Yaskawa INFORM job: R1_W27-A4(90,180)KM-OK.JBI

/JOB
//NAME R1_W27-A4(90,180)KM-OK
///FOLDERNAME KRIS-SCIANA
//POS
///NPOS 201,201,0,9,0,0
///TOOL 0
///POSTYPE PULSE
///PULSE
C00000=-12408,-168229,-129239,11856,76417,1490
C00001=-114075,-55562,-33330,57879,69757,51049
C00002=-170127,-11218,4712,80761,69619,75034
C00003=-166026,1115,14662,80935,66751,75417
C00004=-166026,1115,14662,80935,66751,75417
C00005=-164179,6139,17196,85884,73779,76491
C00006=-163843,5639,16762,85908,73539,76507
C00007=-164179,6139,17196,85884,73779,76491
C00008=-166496,-467,13337,75702,58764,75189
C00009=-166831,-1552,12436,75705,58996,75152
C00010=-166508,-36,14521,75997,58636,74926
C00011=-166831,-1552,12436,75705,58996,75152
C00012=-166496,-467,13337,75702,58764,75189
C00013=-166021,-3570,934,78534,68009,78358
C00014=-137610,-28929,-19421,69080,47942,64710
C00015=-100776,-35686,-23013,57930,21837,49720
C00016=-103071,-36442,-26491,56591,24205,50318
C00017=-97018,-28630,-27379,22144,28331,59500
C00018=-96530,-21499,-20901,21722,27897,59706
C00019=-100662,-29228,-19206,55793,22319,50751
C00020=-102053,-30601,-20713,56706,23278,50281
C00021=-94207,-25966,-26207,14018,29505,61725
C00022=-90744,-41515,-31094,11154,24096,63148
C00023=-90595,-42140,-31027,11070,23720,63189
C00024=-94073,-53021,-44279,15136,26788,61156
C00025=-105496,-45084,-28829,64380,24182,46446
C00026=-120732,-139011,-128731,13191,-67324,-37746
C00027=-120732,-139011,-128731,13191,-67324,-37746
C00028=-21816,-138429,-128213,9073,25992,-35710
C00029=12937,47891,-35883,-5198,71905,46207
C00030=24559,114456,10111,-12521,95879,79421
C00031=-20060,163701,97232,-14944,96585,79331
C00032=-75754,163701,97232,-14944,96585,79331
C00033=-99437,40505,18804,-2837,35585,35366
C00034=-120732,-117814,-48395,13191,72289,-37746
C00035=-172569,-80041,-34226,-15627,55653,-16743
C00036=-173881,-75690,-28267,-15647,54036,-17014
C00037=-174396,-73921,-25835,-15662,53377,-17117
C00038=-174409,-72642,-23726,-15788,52756,-17025
C00039=-174396,-73921,-25835,-15662,53377,-17117
C00040=-177237,-69247,-20992,-27235,53512,-13633
C00041=-177890,-67562,-19632,-27129,53343,-13864
C00042=-177237,-69247,-20992,-27235,53512,-13633
C00043=-181977,-77418,-24251,-27266,50136,-14704
C00044=-193956,-50227,-14941,539,58562,-29056
C00045=-192915,-50819,-15265,329,58451,-28665
C00046=-194756,-48721,-14111,700,58831,-29355
C00047=-182531,-71466,-31778,-1788,58094,-24759
C00048=-122199,17749,55230,-64618,69888,3761
C00049=-124469,25360,65490,-65961,67496,4502
C00050=-125352,28797,70143,-66592,66515,4877
C00051=-125200,39134,82378,-67427,65683,5911
C00052=-125978,39297,82548,-67654,65232,5820
C00053=-125200,39134,82378,-67427,65683,5911
C00054=-125352,28797,70143,-66592,66515,4877
C00055=-127676,20892,69191,-78285,59026,9362
C00056=-127562,25294,74286,-78756,58894,9826
C00057=-127676,21375,69995,-78428,58968,9490
C00058=-125009,20842,69444,-77518,60577,9664
C00059=-122672,36678,78518,-58027,73309,3381
C00060=-122677,38905,82216,-58303,72687,3837
C00061=-122672,36678,78518,-58027,73309,3381
C00062=-172569,-80041,-34226,-15627,55653,-16743
C00063=-193629,-34313,-13531,-412,84628,-47335
C00064=-193629,-29158,-1725,-414,80010,-47323
C00065=-192771,-30731,-2257,-348,79534,-47037
C00066=-192029,-32324,-3298,-290,79358,-46790
C00067=-192512,-31641,-3367,-327,79748,-46950
C00068=-192512,-32314,-4820,-327,80296,-46951
C00069=-191917,-33584,-5641,-280,80152,-46753
C00070=-191917,-33170,-4750,-280,79815,-46753
C00071=-191917,-35734,-10378,-279,81963,-46757
C00072=-120477,17632,43941,-55533,81040,-704
C00073=-135463,1706,26098,-36401,96659,-64397
C00074=-139240,-2239,32183,-37186,90451,-63806
C00075=-139413,-3608,31065,-37238,90369,-63846
C00076=-139240,-2239,32183,-37186,90451,-63806
C00077=-139240,-982,34590,-37167,89779,-63576
C00078=-139240,-2239,32183,-37186,90451,-63806
C00079=-136968,12512,36999,-36743,95104,-64482
C00080=-139711,-16957,6278,-33197,82477,-62153
C00081=-147688,-28677,-1688,-34006,78458,-64099
C00082=-148352,-29126,-1989,-34060,78161,-64273
C00083=-147688,-28677,-1688,-34006,78458,-64099
C00084=-147688,-29352,-3169,-33950,78930,-64245
C00085=-147969,-31758,-4758,-33997,78605,-64257
C00086=-147969,-31405,-3991,-34026,78361,-64182
C00087=-147969,-31758,-4758,-33997,78605,-64257
C00088=-146343,-30027,-3614,-33855,79395,-63850
C00089=-146343,-29533,-2533,-33893,79050,-63746
C00090=-147651,-30771,-3351,-34009,78431,-64078
C00091=-147340,-30313,-4491,-33895,79336,-64232
C00092=-168861,-24308,-1126,-34250,71707,-70597
C00093=-172727,-20891,3494,-34314,69279,-71427
C00094=-173288,-21050,3382,-34292,69050,-71587
C00095=-172727,-20891,3494,-34314,69279,-71427
C00096=-172727,-21623,1837,-34186,69816,-71602
C00097=-173683,-23699,371,-34172,69302,-71836
C00098=-173683,-23301,1270,-34243,69012,-71740
C00099=-173683,-23699,371,-34172,69302,-71836
C00100=-171105,-22755,1033,-34271,70379,-71106
C00101=-171105,-22220,2243,-34361,69988,-70979
C00102=-172969,-22746,1870,-34294,69220,-71509
C00103=-172838,-23509,-311,-34112,70064,-71727
C00104=-172642,-46434,-14047,-37866,50218,-77712
C00105=-173875,-14141,7002,-35805,52648,-79377
C00106=-177522,-4435,19967,-36117,48708,-79612
C00107=-177904,-4485,19925,-35996,48552,-79746
C00108=-177522,-4435,19967,-36117,48708,-79612
C00109=-177522,-5400,17843,-35709,49372,-79894
C00110=-178274,-6796,17094,-35594,48861,-80070
C00111=-178274,-6447,17863,-35742,48620,-79968
C00112=-178274,-6796,17094,-35594,48861,-80070
C00113=-176755,-6519,17315,-36071,49483,-79541
C00114=-176755,-6106,18226,-36244,49200,-79420
C00115=-177745,-6110,18254,-35943,48780,-79759
C00116=-177557,-6572,16647,-35628,49473,-79954
C00117=-127483,-80419,-25529,-45538,63215,-61268
C00118=-137560,-77057,-18811,-45546,71982,-69050
C00119=-137790,-77163,-18085,-45710,71521,-68929
C00120=-138002,-77837,-18318,-45803,71281,-68907
C00121=-137790,-77163,-18085,-45710,71521,-68929
C00122=-137790,-78839,-20640,-45553,72028,-69171
C00123=-138552,-80734,-20734,-45929,71034,-69027
C00124=-138465,-80152,-20160,-45922,71036,-68989
C00125=-138465,-79547,-19253,-45982,70860,-68902
C00126=-138465,-80152,-20160,-45922,71036,-68989
C00127=-130873,-75354,-22667,-43475,77336,-68607
C00128=-143731,-120291,-35892,-61673,37258,-53156
C00129=-153031,-106896,-24772,-72774,26670,-48341
C00130=-154852,-106645,-24753,-72766,25749,-48792
C00131=-174213,-103200,-24560,-67377,16120,-55832
C00132=-173958,-111624,-32831,-65076,16578,-56845
C00133=-173211,-92844,-38044,-39863,60080,-26099
C00134=-183742,-42639,-8543,-30727,93066,-40842
C00135=-194212,-69823,-30460,-23787,74043,-41412
C00136=-189340,-95494,-32602,-40064,42381,-27057
C00137=-199606,-67555,-26283,-19174,46492,-39002
C00138=-192832,-51591,-10291,-33919,35141,-36541
C00139=-193001,-17027,18379,-39421,24969,-38608
C00140=-185793,-2062,15010,-31452,55489,-48604
C00141=-180914,-39023,-11312,-35464,76884,-35483
C00142=-186493,-28244,-7036,-31408,60621,-50185
C00143=-186186,-25103,-332,-32207,58430,-49503
C00144=-187143,4604,23985,-31838,53193,-48465
C00145=-185793,-2062,15010,-31452,55489,-48604
C00146=-188015,-40449,-12502,-32039,52292,-48508
C00147=-190017,-70687,-28062,-34017,46482,-47362
C00148=-197564,-65393,-25632,-20611,46860,-52632
C00149=-193036,-36661,-7528,-24209,47101,-50263
C00150=-187937,-34749,-9314,-31507,53139,-48818
C00151=-174696,-57453,-24242,-35706,56174,-43629
C00152=-140598,-78081,-33659,-39772,66860,-32227
C00153=-141807,-20980,22756,-45396,108405,-42087
C00154=-139242,-49470,8103,-46479,95274,-40803
C00155=-152058,-45207,10125,-51949,89895,-43634
C00156=-147215,-46864,6623,-50076,93094,-43175
C00157=-141782,-45888,-18329,-50852,105894,-47292
C00158=-122197,265,20116,-61362,75919,-1585
C00159=-148312,-18266,18073,-35868,41105,-22148
C00160=-148389,-10811,27499,-37215,39474,-21366
C00161=-148139,-7130,31782,-37859,38978,-20950
C00162=-149047,-9416,30148,-37653,38478,-21229
C00163=-148550,-6621,33826,-38481,38019,-20665
C00164=-151250,-3570,34403,-36506,37914,-22272
C00165=-150396,-8469,29288,-36370,38763,-22201
C00166=-150383,-15985,19712,-34952,40435,-23027
C00167=-136141,-317,34070,-49048,57432,-19039
C00168=-137229,7022,44527,-50381,55121,-18205
C00169=-137621,10190,48745,-50908,54295,-17886
C00170=-137107,11277,51332,-51470,53891,-17317
C00171=-136657,9562,48504,-50983,54669,-17581
C00172=-137398,10846,49256,-50891,54423,-17845
C00173=-137247,10896,49257,-50876,54513,-17818
C00174=-136822,13685,51719,-50910,54678,-17683
C00175=-136799,9316,46568,-50416,55288,-18069
C00176=-135467,4556,38210,-49073,57743,-18855
C00177=-136137,-10257,13643,-45943,62583,-21899
C00178=-136139,-13457,6254,-44950,64655,57340
C00179=-140525,19486,41917,-27486,58532,69458
C00180=-158575,-22743,-5640,-261,63822,52267
C00181=-201270,-72526,-20170,41599,43995,22865
C00182=-208523,-61328,-5512,45049,45103,18922
C00183=-210983,-54521,-945,44398,50079,19814
C00184=-208926,-60351,-4855,45020,45353,18846
C00185=-208139,-60468,-3279,45679,44265,18612
C00186=-209884,-54474,-922,44345,49597,20126
C00187=-202908,-51930,157,43430,46646,22304
C00188=-208516,-61339,-5515,45051,45097,18922
C00189=-207445,-70087,-17224,43111,46602,20424
C00190=-181249,-65588,-30997,-1667,65478,39835
C00191=-185098,-71138,-35276,-1207,65193,38466
C00192=-185098,-71138,-35276,-1207,65193,-61891
C00193=-207460,-36123,-10937,5047,85219,-68239
C00194=-207182,-34469,-3956,5107,81769,-68286
C00195=-200210,-11287,15225,10180,88593,-66064
C00196=-196383,-27179,-3960,6315,84751,-64562
C00197=-180622,-60291,-30151,7915,82491,-59413
C00198=-160502,-110903,-38036,31925,21612,35926
C00199=-124191,-185712,-132113,-18898,16762,67097
C00200=-17783,-160560,-136425,-18898,-7174,67097
BC00000=4712,11801,676331
BC00001=16981,3941,735308
BC00002=144144,15,764761
BC00003=168784,15,764761
BC00004=168784,15,764761
BC00005=169964,15,705864
BC00006=169964,15,705864
BC00007=169964,15,705864
BC00008=192237,15,822054
BC00009=202665,15,821772
BC00010=202665,15,821772
BC00011=202665,15,821772
BC00012=192237,15,822054
BC00013=168784,15,764761
BC00014=111214,15,768197
BC00015=46157,15,772080
BC00016=49226,15,755689
BC00017=50490,16,762582
BC00018=50490,16,762582
BC00019=50454,15,749133
BC00020=50454,15,749133
BC00021=50454,15,749133
BC00022=50454,15,749133
BC00023=50454,15,749133
BC00024=50454,15,749133
BC00025=46195,15,785534
BC00026=143511,1082,90582
BC00027=207222,1082,1056179
BC00028=165072,1082,1056179
BC00029=62550,1470,1070352
BC00030=114350,1997,1074164
BC00031=144804,1997,1074164
BC00032=288140,1997,1074164
BC00033=393476,1653,1067401
BC00034=373932,1082,1056179
BC00035=398174,99453,483906
BC00036=398174,102626,483906
BC00037=398174,103895,483906
BC00038=398174,103895,483906
BC00039=398174,103895,483906
BC00040=398174,123267,483906
BC00041=398174,123392,483906
BC00042=398174,123267,483906
BC00043=398174,123267,483906
BC00044=398174,94527,483906
BC00045=398174,96604,483906
BC00046=398174,94527,483906
BC00047=398174,88092,484425
BC00048=398174,15,483906
BC00049=398174,15,483906
BC00050=398174,15,483906
BC00051=398174,1781,483906
BC00052=398174,1784,483906
BC00053=398174,1781,483906
BC00054=398174,15,483906
BC00055=398174,15,483906
BC00056=398174,15,483906
BC00057=398174,15,483906
BC00058=398174,15,483906
BC00059=398174,17875,483906
BC00060=398174,17501,483906
BC00061=398174,17875,483906
BC00062=398174,99453,483906
BC00063=398174,99453,483906
BC00064=398174,99453,483906
BC00065=398174,99453,483906
BC00066=398174,99453,483906
BC00067=398174,99453,483906
BC00068=398174,99453,483906
BC00069=398174,99453,483906
BC00070=398174,99453,483906
BC00071=398174,99453,483906
BC00072=398174,14811,483906
BC00073=398174,14811,483906
BC00074=398174,14811,483906
BC00075=398174,14811,483906
BC00076=398174,14811,483906
BC00077=398174,14811,483906
BC00078=398174,14811,483906
BC00079=398174,14811,483905
BC00080=398174,14811,882248
BC00081=398174,14811,882248
BC00082=398174,14811,882248
BC00083=398174,14811,882248
BC00084=398174,14811,882248
BC00085=398174,14811,882248
BC00086=398174,14811,882248
BC00087=398174,14811,882248
BC00088=398174,14811,882247
BC00089=398174,14811,882247
BC00090=398174,14811,882247
BC00091=398174,14811,882247
BC00092=398174,73156,882247
BC00093=398174,73156,882247
BC00094=398174,73156,882247
BC00095=398174,73156,882247
BC00096=398174,73156,882247
BC00097=398174,73156,882247
BC00098=398174,73156,882247
BC00099=398174,73156,882247
BC00100=398174,73156,882247
BC00101=398174,73156,882247
BC00102=398174,73156,882247
BC00103=398174,73156,882247
BC00104=398174,73156,882247
BC00105=398174,73156,882247
BC00106=398174,73156,882247
BC00107=398174,73156,882247
BC00108=398174,73156,882247
BC00109=398174,73156,882247
BC00110=398174,73156,882247
BC00111=398174,73156,882247
BC00112=398174,73156,882247
BC00113=398174,73156,882247
BC00114=398174,73156,882247
BC00115=398174,73156,882247
BC00116=398174,73156,882247
BC00117=398174,73156,882247
BC00118=398174,73156,882247
BC00119=398174,73156,882247
BC00120=398174,73156,882247
BC00121=398174,73156,882247
BC00122=398174,73156,882247
BC00123=398174,73156,882247
BC00124=398174,73156,882247
BC00125=398174,73156,882247
BC00126=398174,73156,882247
BC00127=398174,73156,882247
BC00128=398174,73156,882247
BC00129=398174,52305,882247
BC00130=398174,52305,882247
BC00131=398174,52305,882247
BC00132=398174,52305,882247
BC00133=398174,89935,882247
BC00134=398174,89935,882247
BC00135=398174,89935,882247
BC00136=398174,89935,882247
BC00137=398174,89935,882247
BC00138=398174,89935,882247
BC00139=398174,89935,882247
BC00140=398174,89935,882247
BC00141=398174,89935,882247
BC00142=398174,89935,882245
BC00143=398174,89935,882247
BC00144=398174,89935,882247
BC00145=398174,89935,882247
BC00146=398174,89935,882247
BC00147=398174,89935,882247
BC00148=398174,89935,882247
BC00149=398174,89935,882247
BC00150=398174,89935,882247
BC00151=398174,89935,882247
BC00152=398174,89935,882247
BC00153=398174,89935,451645
BC00154=398174,89935,451645
BC00155=398174,89935,451645
BC00156=398174,89935,451645
BC00157=398174,89053,451690
BC00158=398174,15,456194
BC00159=398174,15,483906
BC00160=398174,15,483906
BC00161=398174,15,483906
BC00162=398174,15,483906
BC00163=398174,15,483906
BC00164=398174,15,483906
BC00165=398174,15,483906
BC00166=398174,15,483906
BC00167=398174,15,483906
BC00168=398174,15,483906
BC00169=398174,15,483906
BC00170=398174,15,483906
BC00171=398174,15,483906
BC00172=398174,15,483906
BC00173=398174,3294,483906
BC00174=398174,4443,483906
BC00175=398174,3297,483906
BC00176=398174,433,483906
BC00177=398174,15,472961
BC00178=398174,15,443507
BC00179=398174,15,483906
BC00180=398174,39123,483906
BC00181=398174,96734,483906
BC00182=398174,99364,483906
BC00183=398174,100416,483906
BC00184=398174,100416,483906
BC00185=398174,100416,483906
BC00186=398174,100416,483906
BC00187=398174,100416,483906
BC00188=398174,110550,483906
BC00189=398174,107920,483906
BC00190=398174,107920,483906
BC00191=398174,107920,483906
BC00192=398174,107920,483906
BC00193=398174,107920,483906
BC00194=398174,107920,483906
BC00195=398174,107920,483906
BC00196=398174,107920,483906
BC00197=398174,107920,483906
BC00198=398174,107920,483906
BC00199=398174,107920,1021205
BC00200=2198,23741,1051585
///POSTYPE BASE
///RECTAN
///RCONF 0,0,0,0,1,0,0,0,0,0,0,0,0,0,0,0,0,0,0,0,0,0,0,0
P00006=2.006,1.622,-0.565,0.0000,0.0000,0.0000
P00021=0.073,2.058,-0.109,0.0000,0.0000,0.0000
P00022=2.006,1.622,-0.565,0.0000,0.0000,0.0000
///RCONF 0,0,0,0,0,0,0,0,0,0,0,0,0,0,0,0,0,0,0,0,0,0,0,0
P00023=-2.957,-4.083,2.762,0.0000,0.0000,0.0000
P00024=-1.466,-0.226,-0.419,0.0000,0.0000,0.0000
P00025=3.643,0.007,-2.585,0.0000,0.0000,0.0000
P00026=2.644,0.055,-2.583,0.0000,0.0000,0.0000
P00027=2.278,0.099,-4.210,0.0000,0.0000,0.0000
P00050=-0.123,2.174,-1.314,0.0000,0.0000,0.0000
//INST
///DATE 2025/04/15 14:27
///ATTR SC,RW
///GROUP1 RB1,BS1
NOP
'r1_W27-A4(90,180)
'Path S1000
SFTOF
MOVJ C00000 BC00000 VJ=100.00
MOVJ C00001 BC00001 VJ=100.00
MOVJ C00002 BC00002 VJ=100.00
MOVJ C00003 BC00003 VJ=100.00
MOVL C00004 BC00004 V=166.7
MOVL C00005 BC00005 V=60.0
REFP 3 C00006 BC00006
CALL JOB:SEARCH-R1
SET P023 P006
SFTON P023
MOVL C00007 BC00007 V=60.0
MOVL C00008 BC00008 V=100.0
MOVL C00009 BC00009 V=60.0
REFP 3 C00010 BC00010
CALL JOB:SEARCH-R1
SET P023 P006
SFTON P023
MOVL C00011 BC00011 V=60.0
MOVL C00012 BC00012 V=100.0
'Path VIA1106
SFTOF
MOVJ C00013 BC00013 VJ=20.00
'Path W1001
SFTOF
SFTON P023
MOVJ C00014 BC00014 VJ=20.00
MOVJ C00015 BC00015 VJ=20.00
MOVJ C00016 BC00016 VJ=20.00
MOVL C00017 BC00017 V=166.7 PL=0
MOVL C00018 BC00018 V=83.3
REFP 1 C00019 BC00019
REFP 2 C00020 BC00020
MACRO1 MJ#(0) ARGF7
ARCON
MOVL C00021 BC00021 V=10.8
MOVL C00022 BC00022 V=10.8
MOVL C00023 BC00023 V=10.8
ARCOF
MOVL C00024 BC00024 V=166.7
MOVL C00025 BC00025 V=166.7
SFTOF
'Path VIA1107
SFTOF
MOVJ C00026 BC00026 VJ=40.00
'Path VIA1103
SFTOF
MOVJ C00027 BC00027 VJ=100.00
'Path VIA1104
SFTOF
MOVJ C00028 BC00028 VJ=60.00
MOVJ C00029 BC00029 VJ=30.00
'Path VIA1105
SFTOF
CALL JOB:ONLYCUT-R1_LONG
MOVJ C00030 BC00030 VJ=20.00
MOVJ C00031 BC00031 VJ=40.00
MOVJ C00032 BC00032 VJ=100.00
MOVJ C00033 BC00033 VJ=60.00
SFTOF
MOVJ C00034 BC00034 VJ=80.00
MOVL C00035 BC00035 V=250.0
COMM PAUSE
COMM MOVL C00036 BC00036 V=166.7
COMM MOVL C00037 BC00037 V=60.0
COMM REFP 3 C00038 BC00038
COMM CALL JOB:SEARCH-R1
COMM SET P026 P006
COMM SFTON P026
COMM MOVL C00039 BC00039 V=60.0
COMM MOVL C00040 BC00040 V=60.0
COMM REFP 3 C00041 BC00041
COMM CALL JOB:SEARCH-R1
COMM SET P026 P006
COMM SFTON P026
COMM MOVL C00042 BC00042 V=60.0
COMM MOVL C00043 BC00043 V=100.0
COMM MOVL C00044 BC00044 V=60.0
COMM REFP 3 C00045 BC00045
COMM CALL JOB:SEARCH-R1
COMM SET P026 P006
COMM SFTON P026
COMM MOVL C00046 BC00046 V=60.0
COMM MOVL C00047 BC00047 V=166.7
COMM 'Path S1004
COMM SFTOF
COMM MOVL C00048 BC00048 V=166.7
COMM MOVL C00049 BC00049 V=166.7
COMM MOVL C00050 BC00050 V=100.0
COMM MOVL C00051 BC00051 V=60.0
COMM REFP 3 C00052 BC00052
COMM CALL JOB:SEARCH-R1
COMM SET P027 P006
COMM SFTON P027
COMM MOVL C00053 BC00053 V=60.0
COMM MOVL C00054 BC00054 V=100.0
COMM MOVL C00055 BC00055 V=60.0
COMM REFP 3 C00056 BC00056
COMM CALL JOB:SEARCH-R1
COMM SET P027 P006
COMM SFTON P027
COMM MOVL C00057 BC00057 V=60.0
COMM MOVL C00058 BC00058 V=100.0
COMM MOVL C00059 BC00059 V=60.0
COMM REFP 3 C00060 BC00060
COMM CALL JOB:SEARCH-R1
COMM SET P027 P006
COMM SFTON P027
COMM MOVL C00061 BC00061 V=60.0
COMM PAUSE
MOVJ C00062 BC00062 VJ=100.00
'BP 060624
MOVL C00063 BC00063 V=166.7
MOVL C00064 BC00064 V=166.7
MOVL C00065 BC00065 V=66.7
REFP 3 C00066 BC00066
CALL JOB:SEARCH-R1
SET P050 P006
SFTON P050
MOVL C00067 BC00067 V=60.0
MOVL C00068 BC00068 V=100.0
MOVL C00069 BC00069 V=60.0 PL=0
REFP 3 C00070 BC00070
CALL JOB:SEARCH-R1
SET P050 P006
SFTON P050
MOVL C00071 BC00071 V=60.0
SFTOF
MOVL C00072 BC00072 V=166.7
MOVJ C00073 BC00073 VJ=10.00
MOVL C00074 BC00074 V=66.7
REFP 3 C00075 BC00075
CALL JOB:SEARCH-R1
SET P021 P006
SFTON P021
MOVL C00076 BC00076 V=60.0
REFP 3 C00077 BC00077
CALL JOB:SEARCH-R1
SET P021 P006
SFTON P021
MOVL C00078 BC00078 V=60.0
MOVL C00079 BC00079 V=166.7
MOVL C00080 BC00080 V=250.0
MOVL C00081 BC00081 V=83.3
REFP 3 C00082 BC00082
CALL JOB:SEARCH-R1
SET P022 P006
SFTON P022
MOVL C00083 BC00083 V=60.0
MOVL C00084 BC00084 V=83.3
MOVL C00085 BC00085 V=83.3
REFP 3 C00086 BC00086
CALL JOB:SEARCH-R1
SET P022 P006
SFTON P022
MOVL C00087 BC00087 V=60.0
MOVL C00088 BC00088 V=83.3
MOVL C00089 BC00089 V=83.3
REFP 3 C00090 BC00090
CALL JOB:SEARCH-R1
SET P022 P006
SFTON P022
MOVL C00091 BC00091 V=60.0
MOVL C00092 BC00092 V=166.7
SFTOF
MOVL C00093 BC00093 V=83.3
REFP 3 C00094 BC00094
CALL JOB:SEARCH-R1
SET P023 P006
SFTON P023
MOVL C00095 BC00095 V=100.0
MOVL C00096 BC00096 V=83.3
MOVL C00097 BC00097 V=100.0
REFP 3 C00098 BC00098
CALL JOB:SEARCH-R1
SET P023 P006
SFTON P023
MOVL C00099 BC00099 V=60.0
MOVL C00100 BC00100 V=83.3
MOVL C00101 BC00101 V=100.0
REFP 3 C00102 BC00102
CALL JOB:SEARCH-R1
SET P023 P006
SFTON P023
MOVL C00103 BC00103 V=60.0
MOVL C00104 BC00104 V=100.0
MOVL C00105 BC00105 V=166.7
SFTOF
MOVL C00106 BC00106 V=166.7
REFP 3 C00107 BC00107
CALL JOB:SEARCH-R1
SET P024 P006
SFTON P024
MOVL C00108 BC00108 V=60.0
MOVL C00109 BC00109 V=83.3
MOVL C00110 BC00110 V=83.3
REFP 3 C00111 BC00111
CALL JOB:SEARCH-R1
SET P024 P006
SFTON P024
MOVL C00112 BC00112 V=60.0
MOVL C00113 BC00113 V=83.3
MOVL C00114 BC00114 V=83.3
REFP 3 C00115 BC00115
CALL JOB:SEARCH-R1
SET P024 P006
SFTON P024
MOVL C00116 BC00116 V=60.0
MOVL C00117 BC00117 V=166.7
SFTOF
MOVL C00118 BC00118 V=166.7
MOVL C00119 BC00119 V=166.7
REFP 3 C00120 BC00120
CALL JOB:SEARCH-R1
SET P025 P006
SFTON P025
MOVL C00121 BC00121 V=60.0
MOVL C00122 BC00122 V=166.7
MOVL C00123 BC00123 V=166.7
MOVL C00124 BC00124 V=83.3
REFP 3 C00125 BC00125
CALL JOB:SEARCH-R1
SET P025 P006
SFTON P025
MOVL C00126 BC00126 V=60.0
SFTOF
MOVL C00127 BC00127 V=166.7
MOVL C00128 BC00128 V=166.7
SFTON P025
MACRO1 MJ#(0) ARGF6
MOVL C00129 BC00129 V=166.7
ARCON
MOVL C00130 BC00130 V=11.7
MOVL C00131 BC00131 V=11.7
ARCOF
SFTOF
MOVL C00132 BC00132 V=166.7
MOVL C00133 BC00133 V=166.7
SFTON P022
MACRO1 MJ#(0) ARGF7
MOVL C00134 BC00134 V=166.7 PL=0
ARCON
MOVL C00135 BC00135 V=11.7
MOVL C00136 BC00136 V=11.7
SFTON P023
MOVL C00137 BC00137 V=11.7
MOVL C00138 BC00138 V=11.7
SFTON P024
MOVL C00139 BC00139 V=11.7
ARCOF
MOVL C00140 BC00140 V=166.7
SFTOF
COMM MOVJ C00141 BC00141 VJ=10.00
COMM MOVJ C00142 BC00142 VJ=10.00
COMM SFTON P024
COMM MACRO1 MJ#(0) ARGF7
COMM MOVJ C00143 BC00143 VJ=10.00
COMM ARCON
COMM MOVL C00144 BC00144 V=11.7
COMM ARCOF
COMM MOVJ C00145 BC00145 VJ=10.00
COMM MOVJ C00146 BC00146 VJ=10.00
COMM MOVJ C00147 BC00147 VJ=10.00
COMM SFTOF
COMM SFTON P023
COMM MACRO1 MJ#(0) ARGF7
COMM MOVJ C00148 BC00148 VJ=10.00 PL=0
COMM ARCON
COMM MOVL C00149 BC00149 V=11.7
COMM ARCOF
COMM MOVJ C00150 BC00150 VJ=10.00
COMM SFTOF
MOVJ C00151 BC00151 VJ=10.00
MOVJ C00152 BC00152 VJ=10.00
MOVJ C00153 BC00153 VJ=20.00
SFTON P021
MACRO1 MJ#(0) ARGF7
MOVJ C00154 BC00154 VJ=15.00
ARCON
MOVL C00155 BC00155 V=9.2
ARCOF
MOVJ C00156 BC00156 VJ=10.00
MOVJ C00157 BC00157 VJ=100.00
COMM PAUSE
COMM 'SPAWANIE
COMM 'Path VIA1109
COMM SFTOF
COMM MOVJ C00158 BC00158 VJ=20.00
COMM 'Path W1005
COMM SFTOF
COMM SFTON P026
COMM MOVL C00159 BC00159 V=166.7
COMM MOVL C00160 BC00160 V=166.7
COMM 'COMMENT-SPR
COMM MOVL C00161 BC00161 V=100.0 PL=0
COMM REFP 1 C00162 BC00162
COMM REFP 2 C00163 BC00163
COMM MACRO1 MJ#(0) ARGF7
COMM MOVL C00164 BC00164 V=10.0
COMM ARCOF
COMM MOVL C00165 BC00165 V=166.7
COMM MOVL C00166 BC00166 V=166.7
COMM SFTOF
COMM 'Path W1006
COMM SFTOF
COMM SFTON P026
COMM MOVL C00167 BC00167 V=166.7
COMM MOVL C00168 BC00168 V=166.7
COMM MOVL C00169 BC00169 V=100.0 PL=0
COMM REFP 1 C00170 BC00170
COMM REFP 2 C00171 BC00171
COMM MACRO1 MJ#(0) ARGF7
COMM MOVL C00172 BC00172 V=11.0
COMM MOVL C00173 BC00173 V=11.0
COMM MOVL C00174 BC00174 V=11.0
COMM ARCOF
COMM MOVL C00175 BC00175 V=166.7
COMM MOVL C00176 BC00176 V=166.7
COMM SFTOF
COMM 'Path VIA1110
COMM SFTOF
COMM MOVJ C00177 BC00177 VJ=50.00
COMM 'Path VIA1111
COMM SFTOF
COMM MOVJ C00178 BC00178 VJ=50.00
COMM 'Path W1007
COMM SFTOF
COMM SFTON P026
COMM MOVL C00179 BC00179 V=166.7
COMM MOVJ C00180 BC00180 VJ=20.00
COMM SFTOF
COMM SFTON P027
COMM MOVL C00181 BC00181 V=166.7
COMM MOVL C00182 BC00182 V=166.7
COMM MOVL C00183 BC00183 V=100.0 PL=0
COMM REFP 1 C00184 BC00184
COMM REFP 2 C00185 BC00185
COMM MACRO1 MJ#(0) ARGF9
COMM ARCON
COMM MOVL C00186 BC00186 V=6.7
COMM MOVL C00187 BC00187 V=6.7
COMM ARCOF
COMM MOVL C00188 BC00188 V=166.7
COMM MOVL C00189 BC00189 V=166.7
COMM SFTOF
COMM MOVL C00190 BC00190 V=166.7
COMM MOVJ C00191 BC00191 VJ=50.00
COMM PAUSE
MOVJ C00192 BC00192 VJ=50.00
MOVJ C00193 BC00193 VJ=50.00
SFTON P050
MACRO1 MJ#(0) ARGF7
MOVL C00194 BC00194 V=100.0 PL=0
ARCON
MOVL C00195 BC00195 V=10.8
ARCOF
MOVJ C00196 BC00196 VJ=15.00
SFTOF
MOVJ C00197 BC00197 VJ=50.00
MOVJ C00198 BC00198 VJ=100.00
MOVJ C00199 BC00199 VJ=100.00
MOVJ C00200 BC00200 VJ=50.00
END
